(* IEC 61131-3 sources: 89152_FlorisHendrix_AfstudeerProject/89152_FlorisHendrix_ExamenProject/Stations/Terminal/HMI/Class/PreLoadingScreens, 1 file *)

(* ---- PreLoadingScreens.st ---- *)
(*!
<Class
	Name               = "PreLoadingScreens"
	Revision           = "1.0"
	RealtimeTask       = "false"
	CyclicTask         = "false"
	BackgroundTask     = "false"
	DefBackground      = "10 ms"
	Sigmatek           = "false"
	OSInterface        = "false"
	HighPriority       = "false"
	Automatic          = "false"
	UpdateMode         = "Prescan"
	SharedCommandTable = "true"
	Objectsize         = "(540,180)"
	Comment            = "class for the early screen number enteries">
	<Channels>
		<Server Name="ClassSvr" Visualized="false" Initialize="false" WriteProtected="true" Retentive="false" Comment="class server"/>
	</Channels>
	<RevDoku>
		<Owner Company="Sigmatek"/>
		<Dokumentation Revision="1.0" Date="2020-04-03" Author="PazKem" Company="Sigmatek" Description="Created class - this class has a table which can be upgraded from a user for all screens the user wants to open before the main screen opens"/>
	</RevDoku>
</Class>
*)
PreLoadingScreens : CLASS
  //Servers:
	ClassSvr 	: SvrChCmd_DINT;
  //Clients:
  //Variables:
  //Functions:

	FUNCTION TAB ScreenNumbers;

	FUNCTION VIRTUAL GLOBAL ClassSvr::Read
		VAR_OUTPUT
			output (EAX) 	: DINT;
		END_VAR;
  //Tables:
	FUNCTION @STD
		VAR_OUTPUT
			ret_code	: CONFSTATES;
		END_VAR;
	FUNCTION GLOBAL TAB @CT_;
END_CLASS;

FUNCTION VIRTUAL GLOBAL PreLoadingScreens::ClassSvr::Read
	VAR_OUTPUT
		output (EAX) 	: DINT;
	END_VAR

	output := #ScreenNumbers()$DINT;

END_FUNCTION

FUNCTION TAB PreLoadingScreens::ScreenNumbers
  // In dieser Tabelle werden die Bildschirmnummern eingetragen,
  // welche vor dem Start der Applikation kurz im Hintergrund geöffnet werden.
  // Grund dafür ist zum Beispiel, dass hier Daten aus einem UDC geholt werden müssen.

  // The screen numbers are entered in this table,
  // which are briefly opened in the background before the application is started.
  // The reason for this is, for example, that data must be fetched from a UDC here.

  50250$UDINT,          // Alarme STD Nr
  50300$UDINT,          // EventHistory STD Nr

END_FUNCTION
